(* CODESYS project Tutorial.project

Project tree, tasks and I/O mapping:
  Device : CODESYS Control Win V3 x64, CODESYS, version 3.5.22.30
    application Application
      libraries: Standard, 3.5.22.0 (System)
      task MainTask (cyclic, interval t#20ms, priority 1) calls PLC_PRG
      program PLC_PRG [ST]
      global variables FIO
      Symbols
*)

// Device/Application/FIO
{attribute 'qualified_only'}
VAR_GLOBAL
    iAtEntry 		: BOOL;
    iLowBox 		: BOOL;
    iHighBox 		: BOOL;
    iAtTurnEntry 	: BOOL;
    iAtLoadPos		: BOOL;
    iAtUnloadPos 	: BOOL;
    iAtFront		: BOOL;
    iAtRightEntry	: BOOL;
    iAtLeftEntry	: BOOL;
    iAtRightExit	: BOOL;
    iAtLeftExit		: BOOL;
 
    oFeederConveyor	: BOOL;
    oEntryConveyor 	: BOOL;
    oLoad			: BOOL;
    oUnload			: BOOL;
    oTurn			: BOOL;
    oLeftConveyor	: BOOL;
    oRightConveyor	: BOOL;
END_VAR

// Device/Application/PLC_PRG
PROGRAM PLC_PRG
VAR
	F_AtEntry 			: F_TRIG;
	F_AtTurnEntry 		: F_TRIG;
	F_AtRightEntry		: F_TRIG;
	F_AtLeftEntry		: F_TRIG;
	F_AtRightExit		: F_TRIG;
	F_AtLeftExit		: F_TRIG;
	
	Pallet_on_left		: BOOL := FALSE;
	Pallet_on_right		: BOOL := FALSE;
	Idle 				: BOOL := TRUE;
	Charging			: BOOL := FALSE;
	Turns_charged		: BOOL := FALSE;
	Discharging			: BOOL := FALSE;
	Turns_Discharged	: BOOL := FALSE;
	Turntable_busy		: BOOL := FALSE;
	Discharge_direction : BOOL := FALSE;
	Entry_busy			: BOOL := FALSE;
	Pallet_on_entry		: BOOL := FALSE;
	Count				: WORD := 16#8000;
END_VAR

F_AtEntry(CLK := FIO.iAtEntry);
F_AtTurnEntry(CLK := FIO.iAtTurnEntry);
F_AtRightEntry(CLK := FIO.iAtRightEntry);		           
F_AtLeftEntry(CLK := FIO.iAtLeftEntry);		(* A pallet abandons the turntable, being charged onto the left exit conveyer *)
F_AtRightExit(CLK := FIO.iAtRightExit);
F_AtLeftExit(CLK := FIO.iAtLeftExit); 		(* A pallet abandons the left exit conveyer *)

(**** LEFT EXIT CONVEYER CONTROL ****)
(* Pallet_on_left represents the state of the left exit conveyer: if it carries a pallet, then Pallet_on_left = TRUE *)

IF F_AtLeftExit.Q THEN						(* When a pallet abandons the conveyer *)
	Pallet_on_left := FALSE;				(* Reset Pallet_on_left *)
END_IF;

IF FIO.iAtLeftEntry THEN 					(* When there’s a pallet at the entry of the conveyer *)
	Pallet_on_left := TRUE;					(* Set Pallet_on_left *)
END_IF;

FIO.oLeftConveyor := Pallet_on_left;		(* Left exit conveyer runs for Pallet_on_left = TRUE *)

(**** RIGHT EXIT CONVEYER CONTROL ****)
IF F_AtRightExit.Q THEN  	
	Pallet_on_right := FALSE;
END_IF;

IF FIO.iAtRightEntry THEN		
	Pallet_on_right := TRUE;	
END_IF;

FIO.oRightConveyor := Pallet_on_right;

(**** TURNTABLE CONTROL ****)
IF Idle AND FIO.iAtTurnEntry THEN
	Idle := FALSE;
	Charging := TRUE;
END_IF;

IF Charging AND FIO.iAtFront THEN
	Charging := FALSE;
	Turns_charged := TRUE;	
END_IF;

IF Turns_charged AND FIO.iAtUnloadPos THEN
	Turns_charged := FALSE;
	Discharging := TRUE;
END_IF;

(* The turntable discharges now onto both conveyers. Thus: *)
IF Discharging AND (F_AtRightEntry.Q OR F_AtLeftEntry.Q) THEN
	Discharging := FALSE;
	Turns_Discharged := TRUE;
END_IF;

IF Turns_Discharged AND FIO.iAtLoadPos THEN
	Turns_Discharged := FALSE;
	Idle := TRUE;
END_IF;

IF F_AtTurnEntry.Q THEN  	
	Turntable_busy := TRUE;	
END_IF;

IF Idle THEN  		
	Turntable_busy := FALSE;
END_IF;

(* Computing control outputs according to the current state of the turntable and the direction of the discharge *)
FIO.oLoad := Charging OR Discharging AND Discharge_direction; 
(* Out_2 is TRUE if the discharge is onto the left conveyer *)
FIO.oUnload := Discharging AND NOT Discharge_direction;	   
(* Out_3 is TRUE if the discharge is onto the right conveyer *)
FIO.oTurn := Turns_charged OR Discharging;

(**** ENTRY CONVEYER CONTROL ****)

IF F_AtEntry.Q THEN 			
	Count := ROL (Count,1);		
	IF (Count = WORD#16#2) THEN	
		Entry_busy := TRUE; 			
	END_IF;	
END_IF;

IF F_AtTurnEntry.Q THEN  			
	Discharge_direction := NOT Discharge_direction;

	(** Defining the direction of the discharge: the direction of the discharge changes every time a pallet is discharged from the entry conveyer onto the turntable. If Discharge_direction = FALSE, then the discharge is onto the right conveyer **)

	Entry_busy := FALSE;	 		
	Count := ROR(Count,1); 	
	IF (Count = WORD#16#8000) THEN	
		Pallet_on_entry := FALSE; 			
	END_IF;
END_IF;

IF FIO.iAtEntry THEN		
	Pallet_on_entry := TRUE;	 	
END_IF;
				
FIO.oEntryConveyor := Pallet_on_entry AND (NOT Turntable_busy OR NOT FIO.iAtTurnEntry);	

(**** FEEDING CONVEYER CONTROL ****)
FIO.oFeederConveyor := NOT Entry_busy OR NOT FIO.iAtEntry;

END_PROGRAM
